TEXTLIST FX2TextList
  0 = 'Wait For Fixture Home Pos &  Front Door Open'
  10 = 'Wait For Load1 complete & Door Closed'
  20 = 'Wait For Fixture Clamps Closed '
  30 = 'Wait for Trunion move to Pos2'
  40 = 'Wait for Front Door Open for Second load'
  50 = 'Wait for Load2 Complete & Door Closed'
  60 = 'Wait For Fixture Clamps Closed '
  70 = 'Wait For Trunion move to Pos1 '
  80 = 'Wait for Turntable to move Work Pos'
  90 = 'Wait for Weld Start Cmd to R1 & R2 Robot for First Weld'
  100 = 'Wait for Trunion move to Pos2'
  110 = 'Wait for Weld Start Cmd to R1 & R2 Robot for Second Weld'
  120 = 'Wait For Trunion move to Pos1 For Unload '
  130 = 'Wait For Rear Door Open'
  140 = 'Wait for Unload Start Cmd for R3 Robot'
  150 = 'Wait For Fixture Clamps Opened '
  160 = 'Wait for R3 Robot Pick 1 Complete'
  170 = 'Wait for R3 Robot Move to Pounce'
  180 = 'Wait for Trunion move to Pos2'
  190 = 'Wait For Fixture Clamps Opened '
  200 = 'Wait for R3 Robot Pick 2 Complete'
  210 = 'Wait for Trunion move to Pos1'
  220 = 'Wait For Rear Door Closed'
  230 = 'Wait for R3 Robot Drop 1 Complete'
  240 = 'Wait for R3 Robot Drop 2 Complete'
  250 = 'Wait for Tuntable Rotate to Load Position'
   = ''
END_TEXTLIST

(* stored: Version 1.1.0.1, ProductVersion 3.1.4024.16
   TextList FX2TextList: Id {9a1fcc23-266a-4e12-914d-26fa22161c60} *)
